TYPE EnableXonXoffRx EXTENDS SubIndexModuleBase :
STRUCT
END_STRUCT
END_TYPE

(* stored: Version 1.1.0.1, ProductVersion 3.1.4024.3
   DUT EnableXonXoffRx: Id {1dbcc473-16f8-4f40-b794-66ed5b4d54df} *)
